TYPE ST_DateAndTime :
STRUCT
END_STRUCT
END_TYPE

(* stored: Version 1.1.0.1
   DUT ST_DateAndTime: Id {30f63df5-93f0-4289-bd66-5c3f94d1cc08} *)
